PROGRAM PRG_updateDrives
VAR
END_VAR

GVL_AxisCtrl.Th1_diVeloSet_OUT := GVL_AxisCtrl.Th1_iVeloSet_IN;
GVL_AxisCtrl.Th2_diVeloSet_OUT := GVL_AxisCtrl.Th2_iVeloSet_IN;

END_PROGRAM

(* stored: Version 1.1.0.1, ProductVersion 3.1.4024.2
   POU PRG_updateDrives: Id {bc0ff2d8-d0fd-4873-b659-65a0e940cd4a}, SpecialFunc None *)
